{attribute addProperty BoxType "AT2050-0501-0024"}
{attribute addProperty Id "A_0084_AT2050_5500_0017_AT2050_5500AT2050_C5E5984862678.25"}
{attribute addProperty CRC "2003523927"}
{attribute addProperty SizeInBites "626"}
{attribute addProperty SizeInBytes "78.25"}
TYPE A_0072_AT2050_0501_0024_AT2050_0501_776B5957 EXTENDS AT2050_BA5A9548 :
STRUCT
	{attribute addProperty Name "A_0084_AT2050_5500_0017_AT2050_5500"}
	A_0084_AT2050_5500_0017_AT2050_5500 : AT2050_C5E59848;
END_STRUCT
END_TYPE

(* stored: Version 1.2.0.0, ProductVersion 3.1.4024.9
   DUT A_0072_AT2050_0501_0024_AT2050_0501_776B5957: Id {77d1a365-8d2e-4922-954d-a1b66ac3b6db} *)
